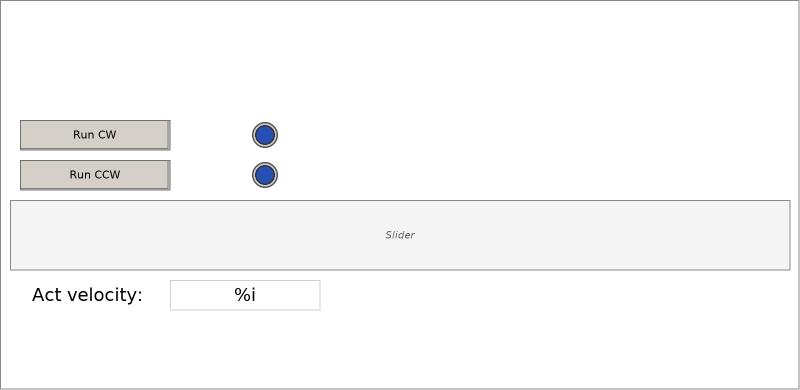
VISUALIZATION VisuAnalogAxisControl  // 800x390
VAR_IN_OUT
	fbManualControler	: FB_ManualController ;
END_VAR
    Slider (10,200 780x70), variable: fbManualControler.pDevAnalogAxis^.stManualCtrl.fCmdVelocity, scale 0..100
    Textfield (170,280 150x30), "%i", text variable: fbManualControler.pDevAnalogAxis^.fActVelocity
        OnMouseClick: write the text variable via VisuDialogs.Numpad
    Label (10,280 150x30), "Act velocity:"
    Button (20,120 150x30), "Run CW"
        tap fbManualControler.pDevAnalogAxis^.stManualCtrl.bCmdRunCW
    Button (20,160 150x30), "Run CCW"
        tap fbManualControler.pDevAnalogAxis^.stManualCtrl.bCmdRunCCW
    Lamp1 (190,120 150x30), variable: fbManualControler.pDevAnalogAxis^.bMovingCW, style: Lamp-Lamp1-Blue
    Lamp1 (190,160 150x30), variable: fbManualControler.pDevAnalogAxis^.bMovingCCW, style: Lamp-Lamp1-Blue
END_VISUALIZATION

(* stored: Version 1.1.0.1, ProductVersion 3.1.4024.11
   Visu VisuAnalogAxisControl: Id {658e100f-f1e3-0cb3-3a0c-4d95fc11e394} *)
